(* Logix 5000 project; controller SX_V040001_C001 vendor 1 type 14 code 77 rev 16.22; software revision 16.04; part 23 of 35 *)
(* tags used below, declared in another part *)
   ALL_KINDS : INT[90];
   CMD : INT[36];
   DRIVE : INT[32];
   EMPTYING : INT[18];
   G_AOutput : DINT[8];
   G_DInput : DINT[3];
   G_DOutput : DINT[3];
   loading : INT[19];
   louvre : INT[11];
   METERING : INT[44];
   PARAMETER : INT[501];
   RM_CMD : INT[9];
   TEMP : INT[14];
(* MainProgram, continued *)

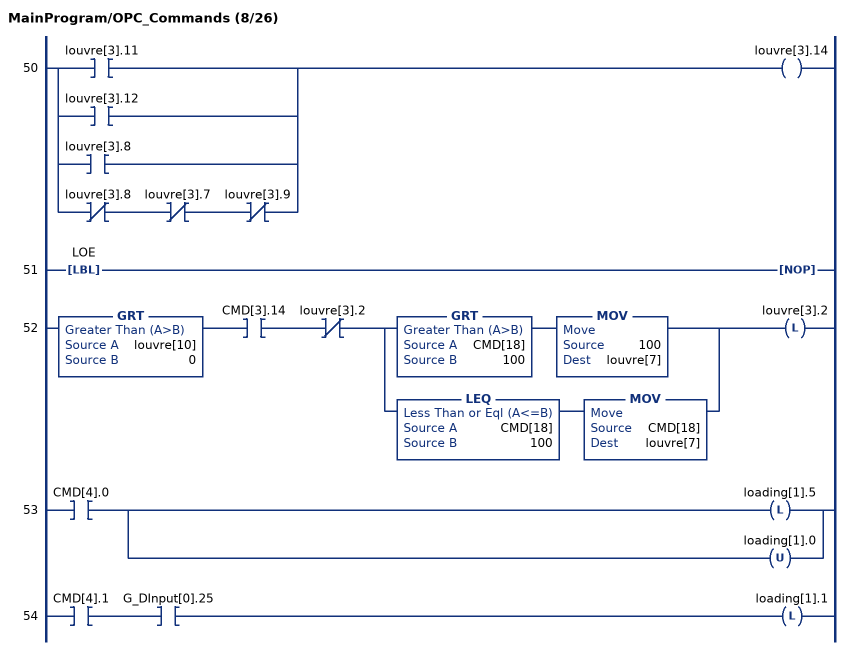
   [picture p501: MainProgram/OPC_Commands rungs 50-54]
   50: [XIC(louvre[3].11) ,XIC(louvre[3].12) ,XIC(louvre[3].8) ,XIO(louvre[3].8) XIO(louvre[3].7) XIO(louvre[3].9) ]OTE(louvre[3].14);
   51: LBL(LOE)NOP();
   52: GRT(louvre[10],0)XIC(CMD[3].14)XIO(louvre[3].2)[GRT(CMD[18],100) MOV(100,louvre[7]) ,LEQ(CMD[18],100) MOV(CMD[18],louvre[7]) ]OTL(louvre[3].2);
   53: XIC(CMD[4].0)[OTL(loading[1].5) ,OTU(loading[1].0) ];
   54: XIC(CMD[4].1)XIC(G_DInput[0].25)OTL(loading[1].1);
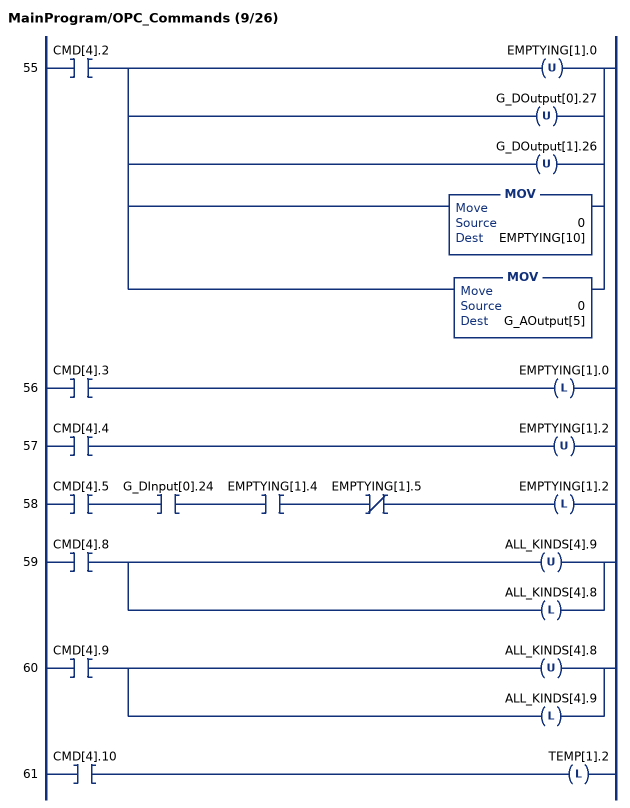
   55: XIC(CMD[4].2)[OTU(EMPTYING[1].0) ,OTU(G_DOutput[0].27) ,OTU(G_DOutput[1].26) ,MOV(0,EMPTYING[10]) ,MOV(0,G_AOutput[5]) ];
   56: XIC(CMD[4].3)OTL(EMPTYING[1].0);
   57: XIC(CMD[4].4)OTU(EMPTYING[1].2);
   58: XIC(CMD[4].5)XIC(G_DInput[0].24)XIC(EMPTYING[1].4)XIO(EMPTYING[1].5)OTL(EMPTYING[1].2);
   59: XIC(CMD[4].8)[OTU(ALL_KINDS[4].9) ,OTL(ALL_KINDS[4].8) ];
   60: XIC(CMD[4].9)[OTU(ALL_KINDS[4].8) ,OTL(ALL_KINDS[4].9) ];
   61: XIC(CMD[4].10)OTL(TEMP[1].2);
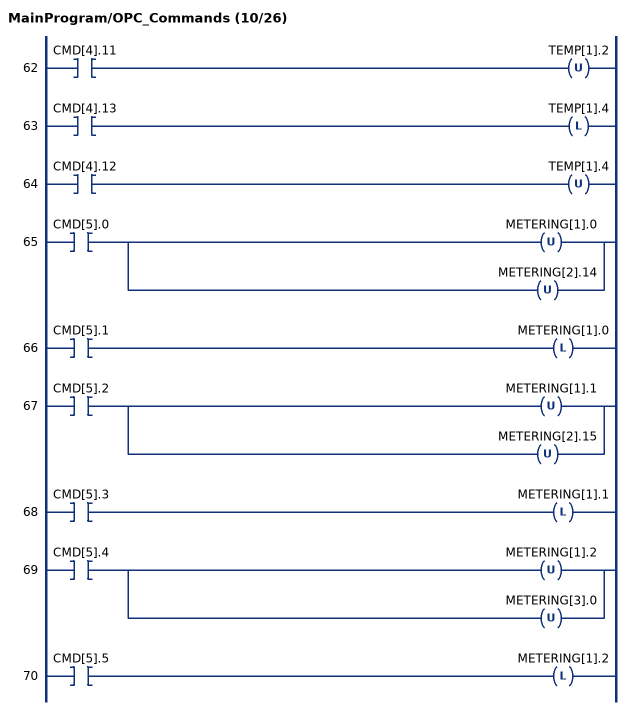
   62: XIC(CMD[4].11)OTU(TEMP[1].2);
   63: XIC(CMD[4].13)OTL(TEMP[1].4);
   64: XIC(CMD[4].12)OTU(TEMP[1].4);
   65: XIC(CMD[5].0)[OTU(METERING[1].0) ,OTU(METERING[2].14) ];
   66: XIC(CMD[5].1)OTL(METERING[1].0);
   67: XIC(CMD[5].2)[OTU(METERING[1].1) ,OTU(METERING[2].15) ];
   68: XIC(CMD[5].3)OTL(METERING[1].1);
   69: XIC(CMD[5].4)[OTU(METERING[1].2) ,OTU(METERING[3].0) ];
   70: XIC(CMD[5].5)OTL(METERING[1].2);
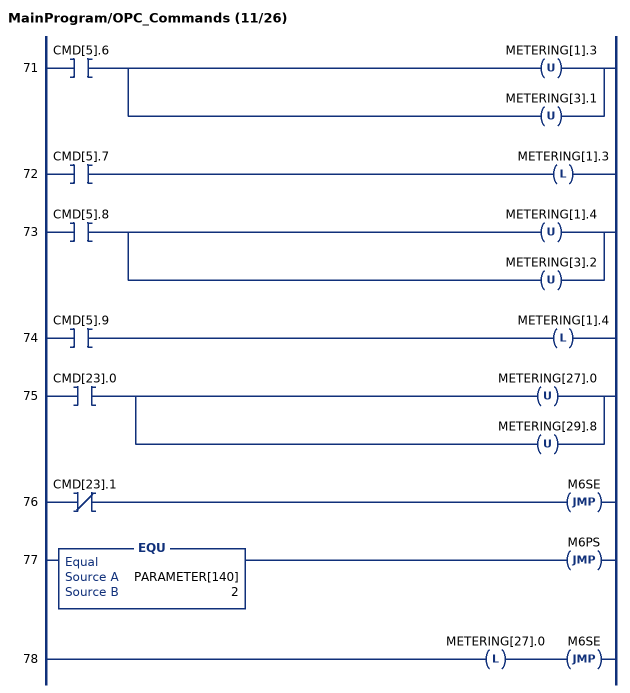
   71: XIC(CMD[5].6)[OTU(METERING[1].3) ,OTU(METERING[3].1) ];
   72: XIC(CMD[5].7)OTL(METERING[1].3);
   73: XIC(CMD[5].8)[OTU(METERING[1].4) ,OTU(METERING[3].2) ];
   74: XIC(CMD[5].9)OTL(METERING[1].4);
   75: XIC(CMD[23].0)[OTU(METERING[27].0) ,OTU(METERING[29].8) ];
   76: XIO(CMD[23].1)JMP(M6SE);
   77: EQU(PARAMETER[140],2)JMP(M6PS);
   78: OTL(METERING[27].0)JMP(M6SE);
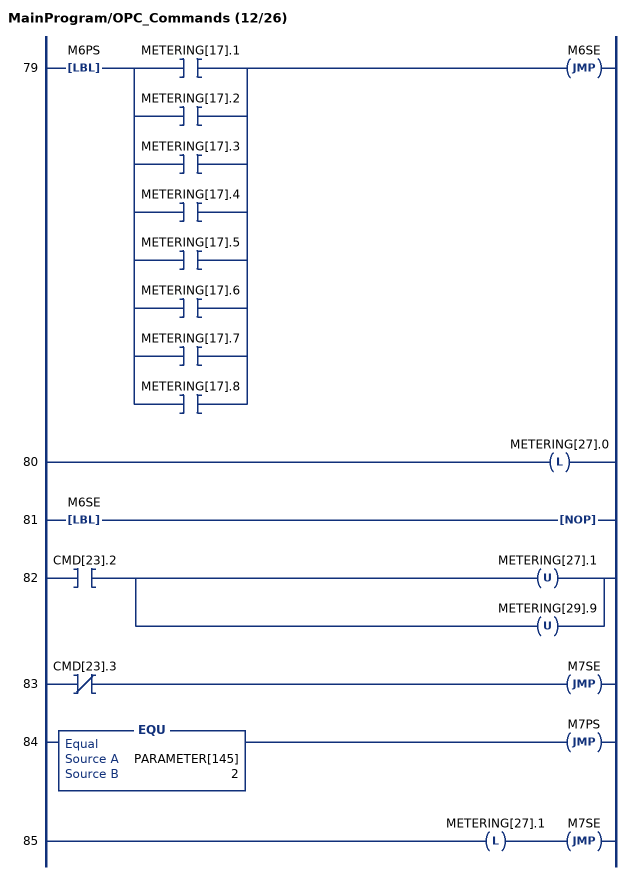
   79: LBL(M6PS)[XIC(METERING[17].1) ,XIC(METERING[17].2) ,XIC(METERING[17].3) ,XIC(METERING[17].4) ,XIC(METERING[17].5) ,XIC(METERING[17].6) ,XIC(METERING[17].7) ,XIC(METERING[17].8) ]JMP(M6SE);
   80: OTL(METERING[27].0);
   81: LBL(M6SE)NOP();
   82: XIC(CMD[23].2)[OTU(METERING[27].1) ,OTU(METERING[29].9) ];
   83: XIO(CMD[23].3)JMP(M7SE);
   84: EQU(PARAMETER[145],2)JMP(M7PS);
   85: OTL(METERING[27].1)JMP(M7SE);
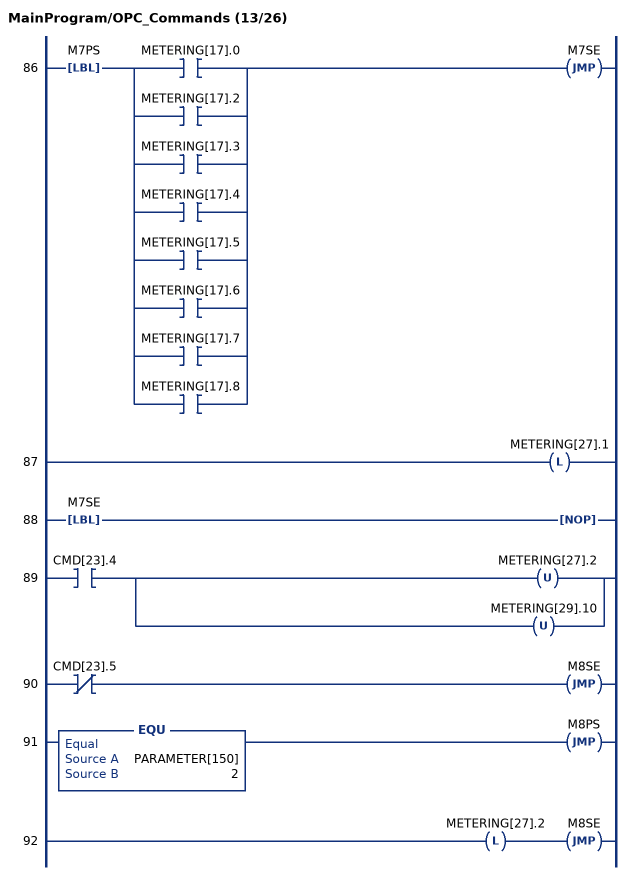
   86: LBL(M7PS)[XIC(METERING[17].0) ,XIC(METERING[17].2) ,XIC(METERING[17].3) ,XIC(METERING[17].4) ,XIC(METERING[17].5) ,XIC(METERING[17].6) ,XIC(METERING[17].7) ,XIC(METERING[17].8) ]JMP(M7SE);
   87: OTL(METERING[27].1);
   88: LBL(M7SE)NOP();
   89: XIC(CMD[23].4)[OTU(METERING[27].2) ,OTU(METERING[29].10) ];
   90: XIO(CMD[23].5)JMP(M8SE);
   91: EQU(PARAMETER[150],2)JMP(M8PS);
   92: OTL(METERING[27].2)JMP(M8SE);
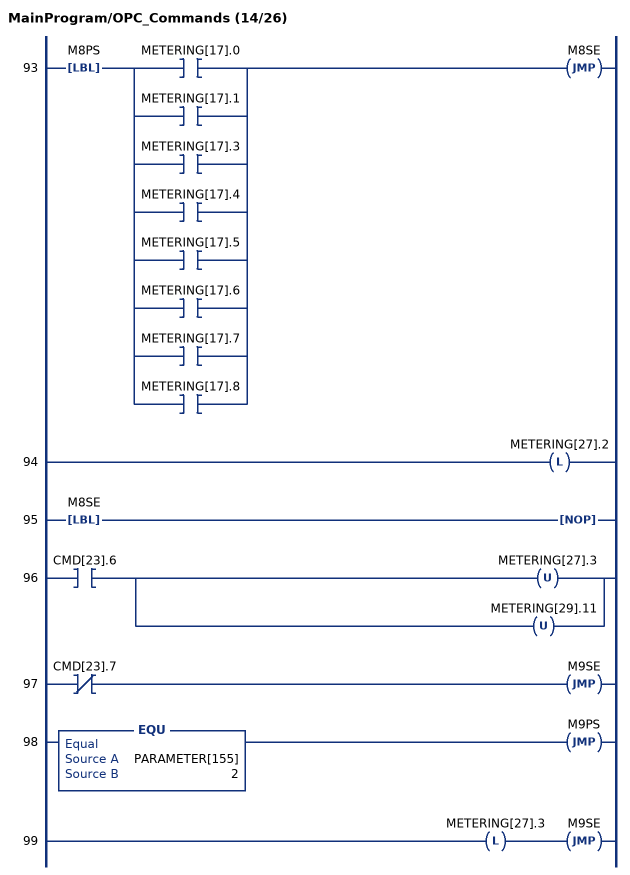
   93: LBL(M8PS)[XIC(METERING[17].0) ,XIC(METERING[17].1) ,XIC(METERING[17].3) ,XIC(METERING[17].4) ,XIC(METERING[17].5) ,XIC(METERING[17].6) ,XIC(METERING[17].7) ,XIC(METERING[17].8) ]JMP(M8SE);
   94: OTL(METERING[27].2);
   95: LBL(M8SE)NOP();
   96: XIC(CMD[23].6)[OTU(METERING[27].3) ,OTU(METERING[29].11) ];
   97: XIO(CMD[23].7)JMP(M9SE);
   98: EQU(PARAMETER[155],2)JMP(M9PS);
   99: OTL(METERING[27].3)JMP(M9SE);
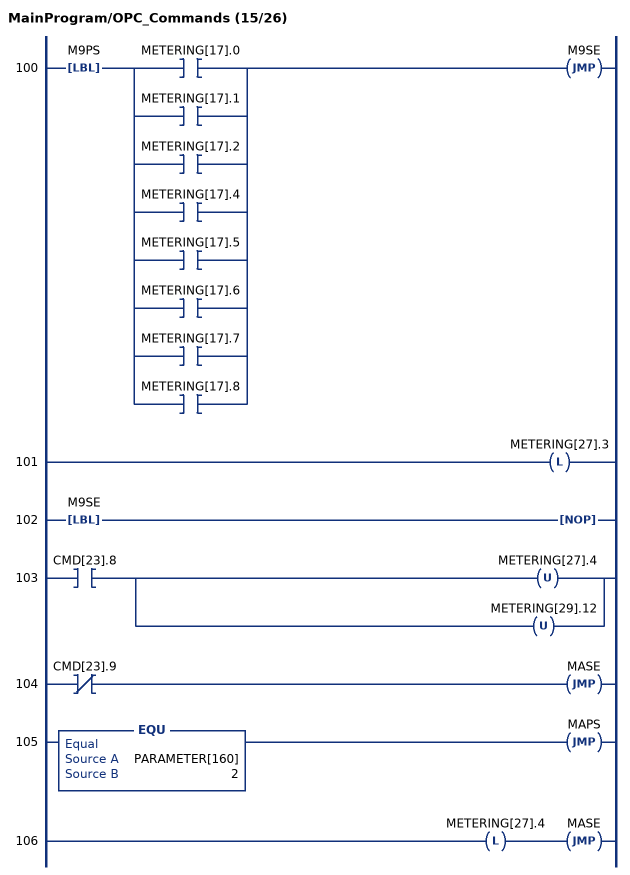
   100: LBL(M9PS)[XIC(METERING[17].0) ,XIC(METERING[17].1) ,XIC(METERING[17].2) ,XIC(METERING[17].4) ,XIC(METERING[17].5) ,XIC(METERING[17].6) ,XIC(METERING[17].7) ,XIC(METERING[17].8) ]JMP(M9SE);
   101: OTL(METERING[27].3);
   102: LBL(M9SE)NOP();
   103: XIC(CMD[23].8)[OTU(METERING[27].4) ,OTU(METERING[29].12) ];
   104: XIO(CMD[23].9)JMP(MASE);
   105: EQU(PARAMETER[160],2)JMP(MAPS);
   106: OTL(METERING[27].4)JMP(MASE);
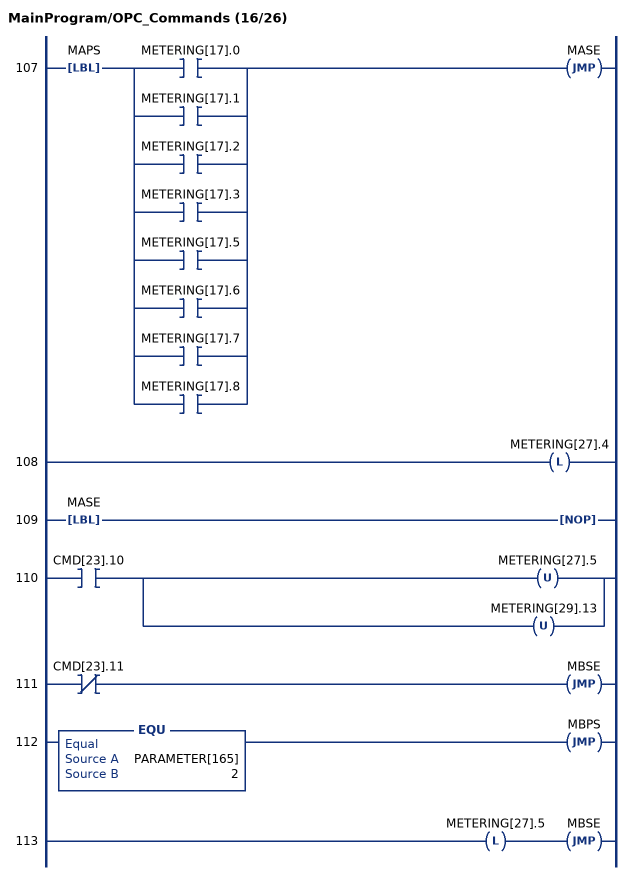
   107: LBL(MAPS)[XIC(METERING[17].0) ,XIC(METERING[17].1) ,XIC(METERING[17].2) ,XIC(METERING[17].3) ,XIC(METERING[17].5) ,XIC(METERING[17].6) ,XIC(METERING[17].7) ,XIC(METERING[17].8) ]JMP(MASE);
   108: OTL(METERING[27].4);
   109: LBL(MASE)NOP();
   110: XIC(CMD[23].10)[OTU(METERING[27].5) ,OTU(METERING[29].13) ];
   111: XIO(CMD[23].11)JMP(MBSE);
   112: EQU(PARAMETER[165],2)JMP(MBPS);
   113: OTL(METERING[27].5)JMP(MBSE);
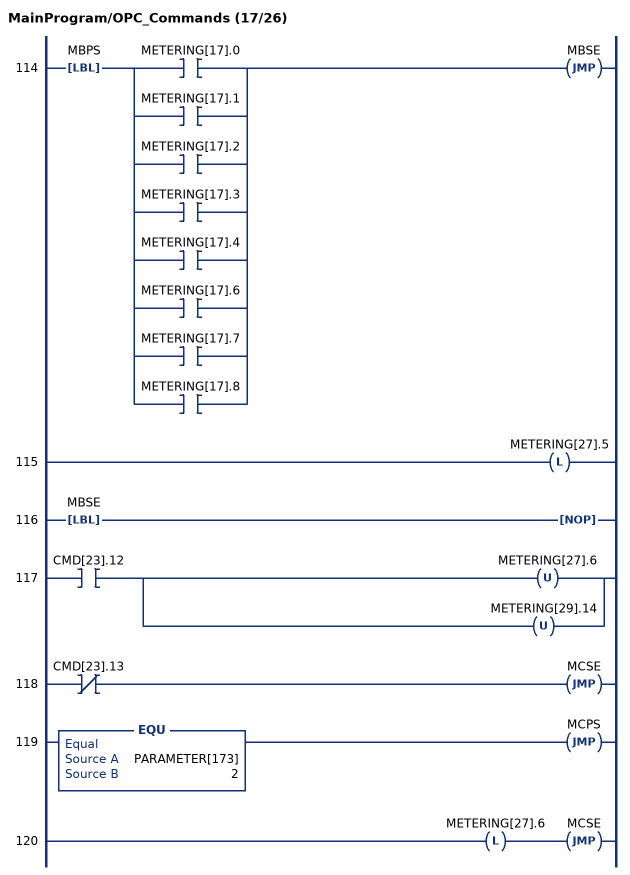
   114: LBL(MBPS)[XIC(METERING[17].0) ,XIC(METERING[17].1) ,XIC(METERING[17].2) ,XIC(METERING[17].3) ,XIC(METERING[17].4) ,XIC(METERING[17].6) ,XIC(METERING[17].7) ,XIC(METERING[17].8) ]JMP(MBSE);
   115: OTL(METERING[27].5);
   116: LBL(MBSE)NOP();
   117: XIC(CMD[23].12)[OTU(METERING[27].6) ,OTU(METERING[29].14) ];
   118: XIO(CMD[23].13)JMP(MCSE);
   119: EQU(PARAMETER[173],2)JMP(MCPS);
   120: OTL(METERING[27].6)JMP(MCSE);
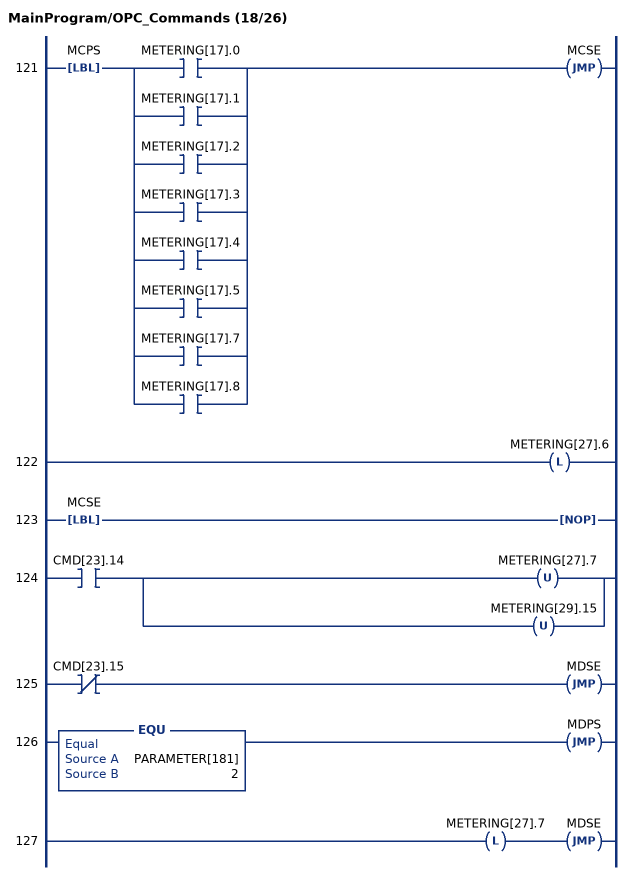
   121: LBL(MCPS)[XIC(METERING[17].0) ,XIC(METERING[17].1) ,XIC(METERING[17].2) ,XIC(METERING[17].3) ,XIC(METERING[17].4) ,XIC(METERING[17].5) ,XIC(METERING[17].7) ,XIC(METERING[17].8) ]JMP(MCSE);
   122: OTL(METERING[27].6);
   123: LBL(MCSE)NOP();
   124: XIC(CMD[23].14)[OTU(METERING[27].7) ,OTU(METERING[29].15) ];
   125: XIO(CMD[23].15)JMP(MDSE);
   126: EQU(PARAMETER[181],2)JMP(MDPS);
   127: OTL(METERING[27].7)JMP(MDSE);
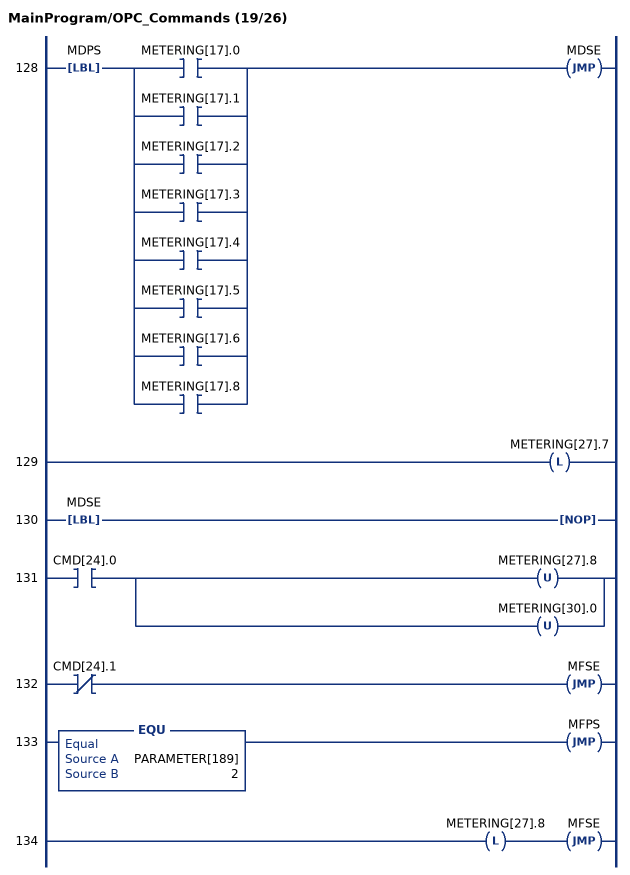
   128: LBL(MDPS)[XIC(METERING[17].0) ,XIC(METERING[17].1) ,XIC(METERING[17].2) ,XIC(METERING[17].3) ,XIC(METERING[17].4) ,XIC(METERING[17].5) ,XIC(METERING[17].6) ,XIC(METERING[17].8) ]JMP(MDSE);
   129: OTL(METERING[27].7);
   130: LBL(MDSE)NOP();
   131: XIC(CMD[24].0)[OTU(METERING[27].8) ,OTU(METERING[30].0) ];
   132: XIO(CMD[24].1)JMP(MFSE);
   133: EQU(PARAMETER[189],2)JMP(MFPS);
   134: OTL(METERING[27].8)JMP(MFSE);
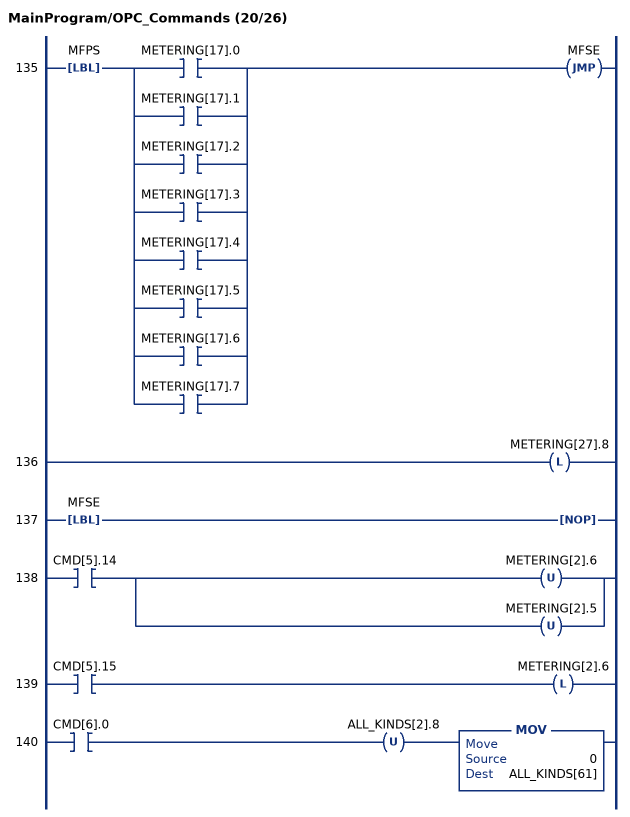
   135: LBL(MFPS)[XIC(METERING[17].0) ,XIC(METERING[17].1) ,XIC(METERING[17].2) ,XIC(METERING[17].3) ,XIC(METERING[17].4) ,XIC(METERING[17].5) ,XIC(METERING[17].6) ,XIC(METERING[17].7) ]JMP(MFSE);
   136: OTL(METERING[27].8);
   137: LBL(MFSE)NOP();
   138: XIC(CMD[5].14)[OTU(METERING[2].6) ,OTU(METERING[2].5) ];
   139: XIC(CMD[5].15)OTL(METERING[2].6);
   140: XIC(CMD[6].0)OTU(ALL_KINDS[2].8)MOV(0,ALL_KINDS[61]);
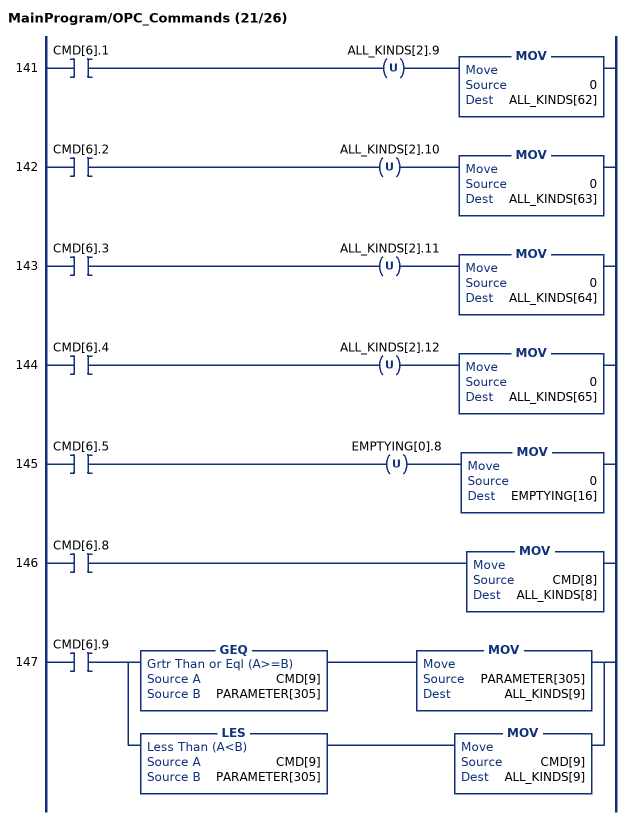
   141: XIC(CMD[6].1)OTU(ALL_KINDS[2].9)MOV(0,ALL_KINDS[62]);
   142: XIC(CMD[6].2)OTU(ALL_KINDS[2].10)MOV(0,ALL_KINDS[63]);
   143: XIC(CMD[6].3)OTU(ALL_KINDS[2].11)MOV(0,ALL_KINDS[64]);
   144: XIC(CMD[6].4)OTU(ALL_KINDS[2].12)MOV(0,ALL_KINDS[65]);
   145: XIC(CMD[6].5)OTU(EMPTYING[0].8)MOV(0,EMPTYING[16]);
   146: XIC(CMD[6].8)MOV(CMD[8],ALL_KINDS[8]);
   147: XIC(CMD[6].9)[GEQ(CMD[9],PARAMETER[305]) MOV(PARAMETER[305],ALL_KINDS[9]) ,LES(CMD[9],PARAMETER[305]) MOV(CMD[9],ALL_KINDS[9]) ];
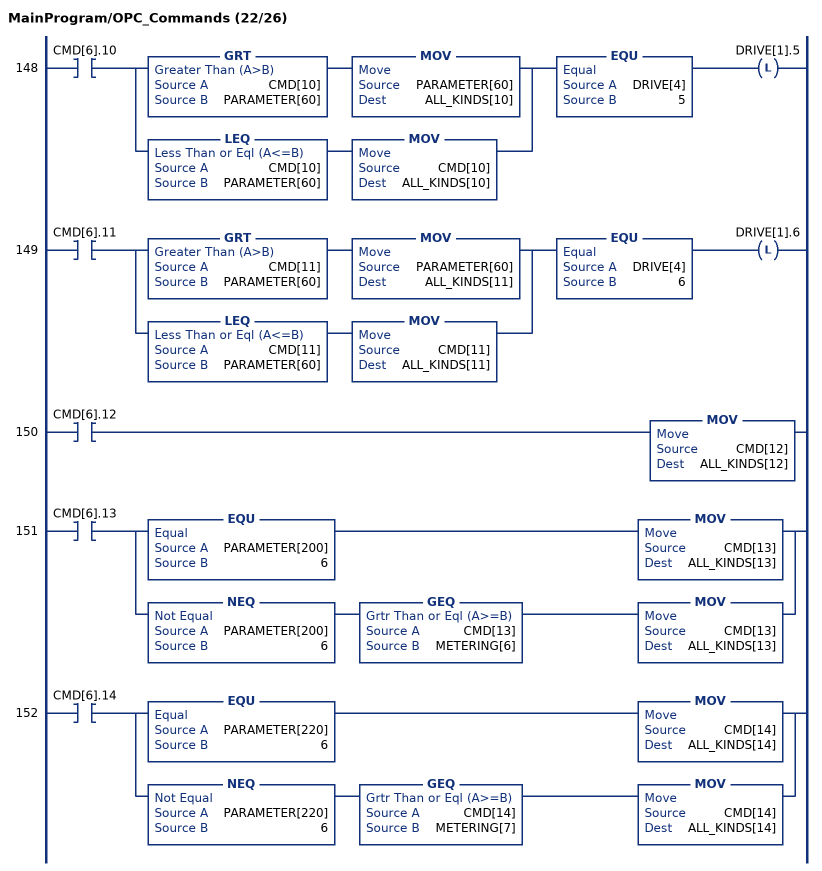
   148: XIC(CMD[6].10)[GRT(CMD[10],PARAMETER[60]) MOV(PARAMETER[60],ALL_KINDS[10]) ,LEQ(CMD[10],PARAMETER[60]) MOV(CMD[10],ALL_KINDS[10]) ]EQU(DRIVE[4],5)OTL(DRIVE[1].5);
   149: XIC(CMD[6].11)[GRT(CMD[11],PARAMETER[60]) MOV(PARAMETER[60],ALL_KINDS[11]) ,LEQ(CMD[11],PARAMETER[60]) MOV(CMD[11],ALL_KINDS[11]) ]EQU(DRIVE[4],6)OTL(DRIVE[1].6);
   150: XIC(CMD[6].12)MOV(CMD[12],ALL_KINDS[12]);
   151: XIC(CMD[6].13)[EQU(PARAMETER[200],6) MOV(CMD[13],ALL_KINDS[13]) ,NEQ(PARAMETER[200],6) GEQ(CMD[13],METERING[6]) MOV(CMD[13],ALL_KINDS[13]) ];
   152: XIC(CMD[6].14)[EQU(PARAMETER[220],6) MOV(CMD[14],ALL_KINDS[14]) ,NEQ(PARAMETER[220],6) GEQ(CMD[14],METERING[7]) MOV(CMD[14],ALL_KINDS[14]) ];
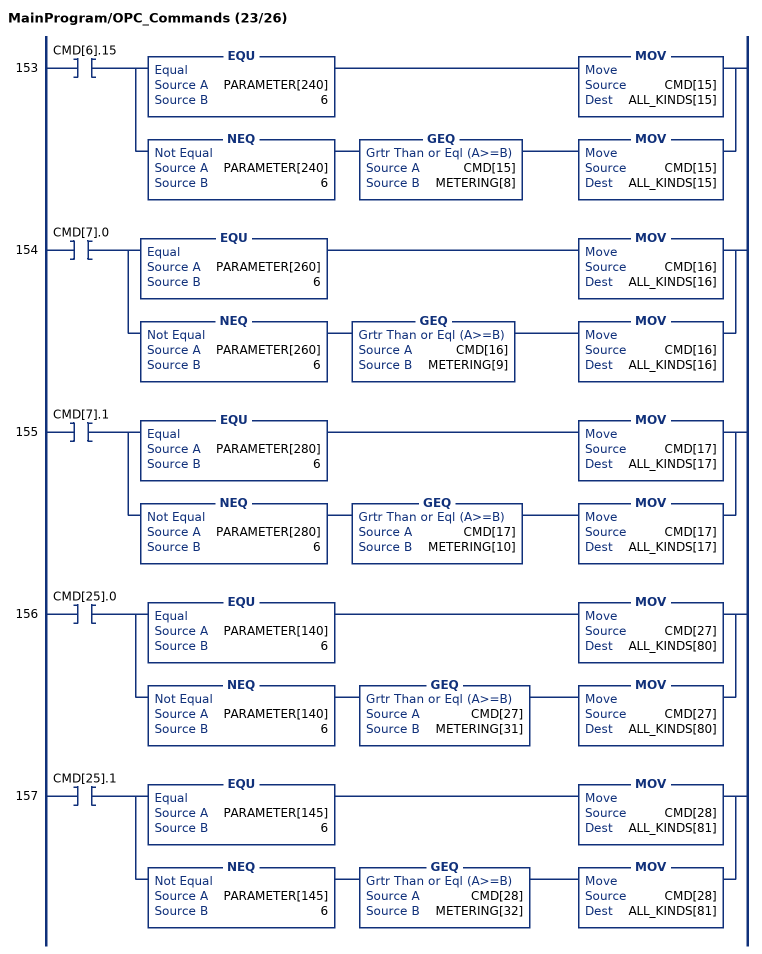
   153: XIC(CMD[6].15)[EQU(PARAMETER[240],6) MOV(CMD[15],ALL_KINDS[15]) ,NEQ(PARAMETER[240],6) GEQ(CMD[15],METERING[8]) MOV(CMD[15],ALL_KINDS[15]) ];
   154: XIC(CMD[7].0)[EQU(PARAMETER[260],6) MOV(CMD[16],ALL_KINDS[16]) ,NEQ(PARAMETER[260],6) GEQ(CMD[16],METERING[9]) MOV(CMD[16],ALL_KINDS[16]) ];
   155: XIC(CMD[7].1)[EQU(PARAMETER[280],6) MOV(CMD[17],ALL_KINDS[17]) ,NEQ(PARAMETER[280],6) GEQ(CMD[17],METERING[10]) MOV(CMD[17],ALL_KINDS[17]) ];
   156: XIC(CMD[25].0)[EQU(PARAMETER[140],6) MOV(CMD[27],ALL_KINDS[80]) ,NEQ(PARAMETER[140],6) GEQ(CMD[27],METERING[31]) MOV(CMD[27],ALL_KINDS[80]) ];
   157: XIC(CMD[25].1)[EQU(PARAMETER[145],6) MOV(CMD[28],ALL_KINDS[81]) ,NEQ(PARAMETER[145],6) GEQ(CMD[28],METERING[32]) MOV(CMD[28],ALL_KINDS[81]) ];
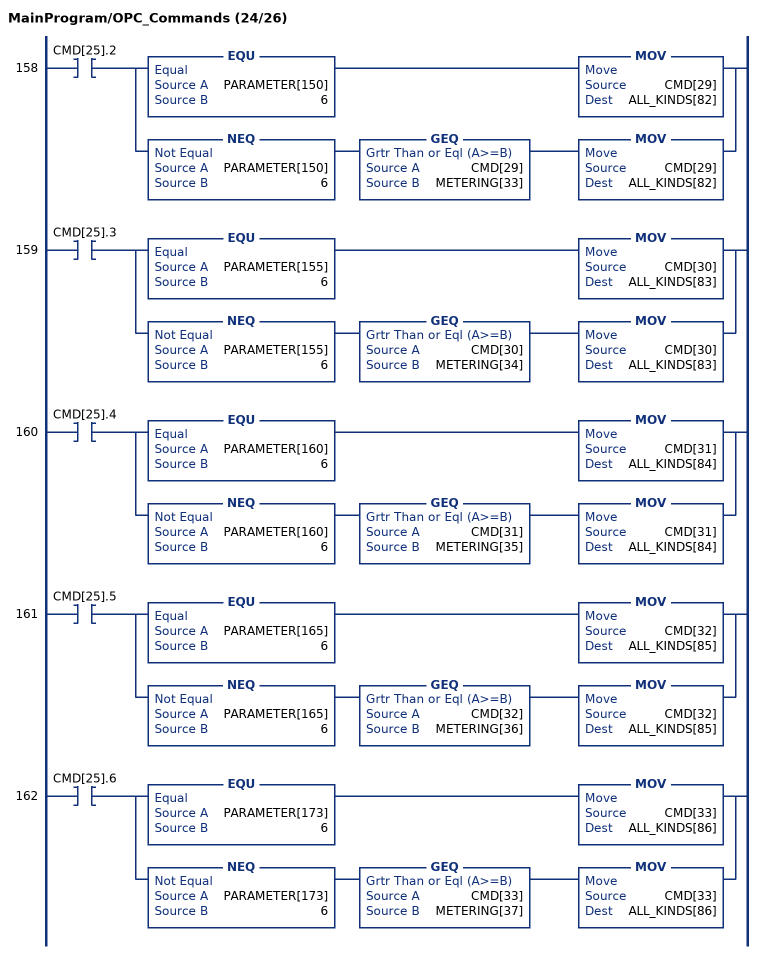
   158: XIC(CMD[25].2)[EQU(PARAMETER[150],6) MOV(CMD[29],ALL_KINDS[82]) ,NEQ(PARAMETER[150],6) GEQ(CMD[29],METERING[33]) MOV(CMD[29],ALL_KINDS[82]) ];
   159: XIC(CMD[25].3)[EQU(PARAMETER[155],6) MOV(CMD[30],ALL_KINDS[83]) ,NEQ(PARAMETER[155],6) GEQ(CMD[30],METERING[34]) MOV(CMD[30],ALL_KINDS[83]) ];
   160: XIC(CMD[25].4)[EQU(PARAMETER[160],6) MOV(CMD[31],ALL_KINDS[84]) ,NEQ(PARAMETER[160],6) GEQ(CMD[31],METERING[35]) MOV(CMD[31],ALL_KINDS[84]) ];
   161: XIC(CMD[25].5)[EQU(PARAMETER[165],6) MOV(CMD[32],ALL_KINDS[85]) ,NEQ(PARAMETER[165],6) GEQ(CMD[32],METERING[36]) MOV(CMD[32],ALL_KINDS[85]) ];
   162: XIC(CMD[25].6)[EQU(PARAMETER[173],6) MOV(CMD[33],ALL_KINDS[86]) ,NEQ(PARAMETER[173],6) GEQ(CMD[33],METERING[37]) MOV(CMD[33],ALL_KINDS[86]) ];
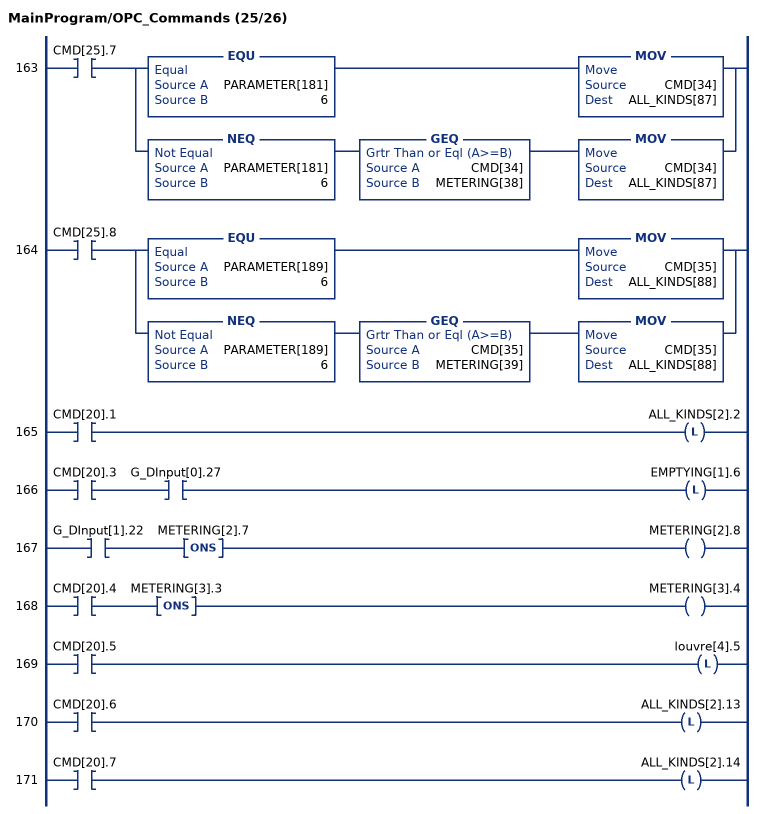
   163: XIC(CMD[25].7)[EQU(PARAMETER[181],6) MOV(CMD[34],ALL_KINDS[87]) ,NEQ(PARAMETER[181],6) GEQ(CMD[34],METERING[38]) MOV(CMD[34],ALL_KINDS[87]) ];
   164: XIC(CMD[25].8)[EQU(PARAMETER[189],6) MOV(CMD[35],ALL_KINDS[88]) ,NEQ(PARAMETER[189],6) GEQ(CMD[35],METERING[39]) MOV(CMD[35],ALL_KINDS[88]) ];
   165: XIC(CMD[20].1)OTL(ALL_KINDS[2].2);
   166: XIC(CMD[20].3)XIC(G_DInput[0].27)OTL(EMPTYING[1].6);
   167: XIC(G_DInput[1].22)ONS(METERING[2].7)OTE(METERING[2].8);
   168: XIC(CMD[20].4)ONS(METERING[3].3)OTE(METERING[3].4);
   169: XIC(CMD[20].5)OTL(louvre[4].5);
   170: XIC(CMD[20].6)OTL(ALL_KINDS[2].13);
   171: XIC(CMD[20].7)OTL(ALL_KINDS[2].14);
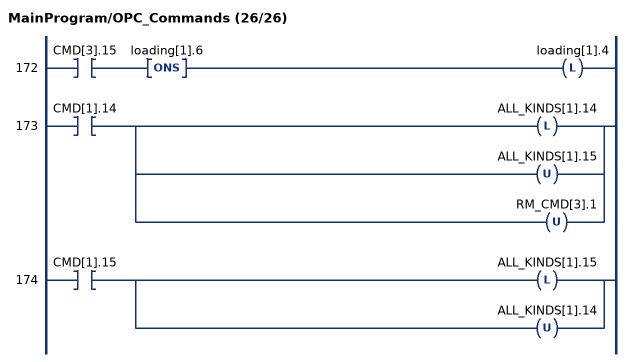
   172: XIC(CMD[3].15)ONS(loading[1].6)OTL(loading[1].4);
   173: XIC(CMD[1].14)[OTL(ALL_KINDS[1].14) ,OTU(ALL_KINDS[1].15) ,OTU(RM_CMD[3].1) ];
   174: XIC(CMD[1].15)[OTL(ALL_KINDS[1].15) ,OTU(ALL_KINDS[1].14) ];
END_ROUTINE
